% RSLogix 500 project PROC1_PID_HEATER_CONTROL.RSS, saved by version 8.30.00.16 %
PROJECT "PROC1"    % processor: Bul.1763 MicroLogix 1100 Series B %

PROGRAM FILES
  LAD 2 "MAIN"  2 rungs
  LAD 3 "IO"  5 rungs
  LAD 4 "PID CNTRL"  4 rungs

DATA FILES
  O0 OUTPUT  9 elements
  I1 INPUT  16 elements
  S2 STATUS  66 elements
  B3 BINARY  1 elements
  T4 TIMER  2 elements
  C5 COUNTER  1 elements
  R6 CONTROL  1 elements
  N7 INTEGER  2 elements
  F8 FLOAT  1 elements
  PD9 TEMP  1 elements

LADDER 2 "MAIN"
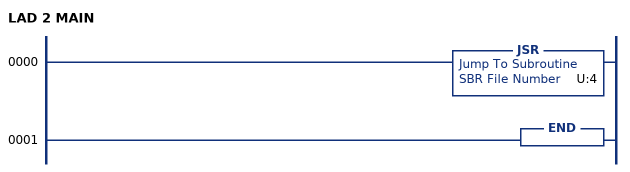
% Rung: 0 %
SOR JSR U:4 EOR
% Rung: 1 %
SOR END EOR

LADDER 3 "IO"
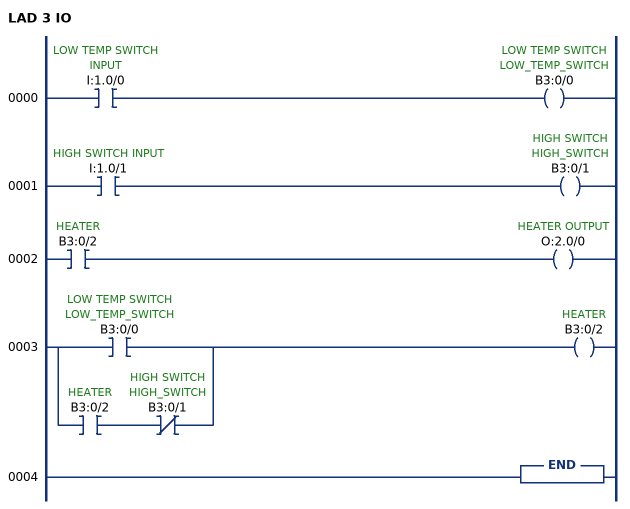
% Rung: 0 %
SOR XIC I:1.0/0 OTE B3:0/0 EOR
%   I:1.0/0  "LOW TEMP SWITCH INPUT" %
%   B3:0/0  LOW_TEMP_SWITCH  "LOW TEMP SWITCH" %
% Rung: 1 %
SOR XIC I:1.0/1 OTE B3:0/1 EOR
%   I:1.0/1  "HIGH SWITCH INPUT" %
%   B3:0/1  HIGH_SWITCH  "HIGH SWITCH" %
% Rung: 2 %
SOR XIC B3:0/2 OTE O:2.0/0 EOR
%   B3:0/2  "HEATER" %
%   O:2.0/0  "HEATER OUTPUT" %
% Rung: 3 %
SOR BST XIC B3:0/0 NXB XIC B3:0/2 XIO B3:0/1 BND OTE B3:0/2 EOR
%   B3:0/0  LOW_TEMP_SWITCH  "LOW TEMP SWITCH" %
%   B3:0/2  "HEATER" %
%   B3:0/1  HIGH_SWITCH  "HIGH SWITCH" %
% Rung: 4 %
SOR END EOR

LADDER 4 "PID CNTRL"
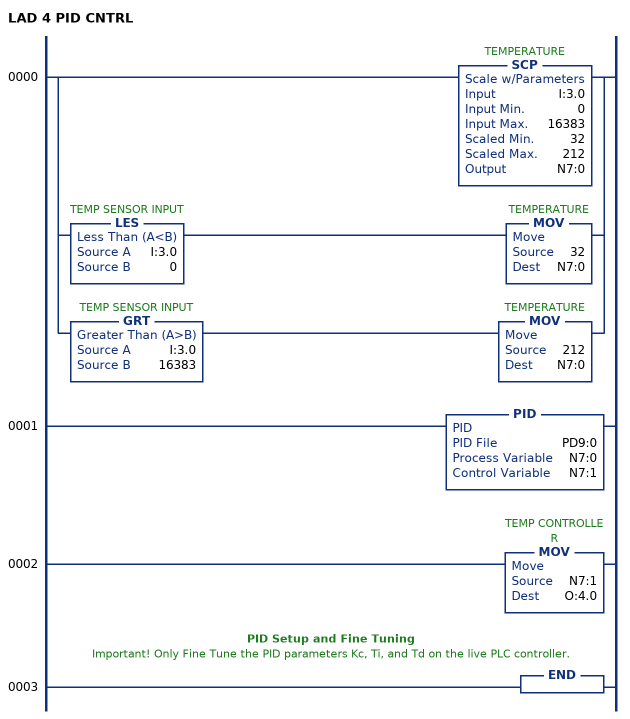
% Rung: 0 %
SOR BST SCP I:3.0 0 16383 32 212 N7:0 NXB LES I:3.0 0 MOV 32 N7:0 NXB GRT I:3.0 16383 MOV 212 N7:0 BND EOR
%   I:3.0  "TEMP SENSOR INPUT" %
%   N7:0  "TEMPERATURE" %
% Rung: 1 %
SOR PID PD9:0 N7:0 N7:1 EOR
%   N7:0  "TEMPERATURE" %
%   N7:1  "PID OUTPUT" %
% Rung: 2 %
SOR MOV N7:1 O:4.0 EOR
%   N7:1  "PID OUTPUT" %
%   O:4.0  "TEMP CONTROLLER" %
% Rung: 3 %
% TITLE: PID Setup and Fine Tuning %
% Important! Only Fine Tune the PID parameters Kc, Ti, and Td on the live PLC controller. %
SOR END EOR

OTHER DOCUMENTED ADDRESSES
  B3:0/3  HH_SWITCH  "HH SWITCH"
  B3:0/4  PUMP  "PUMP"
  B3:0/5  VALVE  "VALVE"
  B3:0/6  FILL_MODE  "FILL MODE = 1 DRAIN MODE = 0"
  I:1.0/2  "H SWITCH INPUT"
  I:1.0/3  "HH SWITCH INPUT"
  O:2.0/1  "PUMP"
  PD9  
  T4:0  "FILL MODE DELAY TIMER"
  T4:1  "DRAIN MODE DELAY TIMER"

REVISION NOTES
  0: Added analog IO
  1: Added PID Logic
  2: Added TEMP Sensor checks

DATA TABLE (non-zero values as saved)
DATA T4
% .PRE .ACC %
% T4:0 % 10 0
% T4:1 % 10 0
